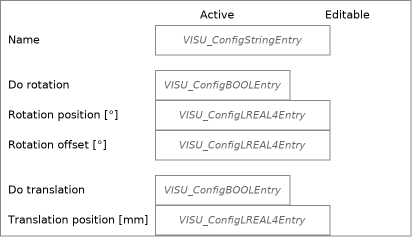
VISUALIZATION VISU_M3Config_KnownPosition  // 412x237
VAR_IN_OUT
	active : M3PositionConfig;
	editable : M3PositionConfig;
END_VAR
    Label (155,5 125x20), "Active"
    Label (285,5 125x20), "Editable"
    Label (5,25 125x30), "Name"
    Frame (155,25 175x30)
        shows VISU_ConfigStringEntry(active := active.name, editable := editable.name)
    Label (5,70 125x30), "Do rotation"
    Frame (155,70 135x30)
        shows VISU_ConfigBOOLEntry(active := active.doRotation, editable := editable.doRotation)
    Frame (155,100 175x30)
        shows VISU_ConfigLREAL4Entry(active := active.rotationPosition, editable := editable.rotationPosition)
    Label (5,100 125x30), "Rotation position [°]"
    Label (5,130 125x30), "Rotation offset [°]"
    Frame (155,130 175x30)
        shows VISU_ConfigLREAL4Entry(active := active.rotationOffset, editable := editable.rotationOffset)
    Label (5,175 125x30), "Do translation"
    Frame (155,175 135x30)
        shows VISU_ConfigBOOLEntry(active := active.doTranslation, editable := editable.doTranslation)
    Frame (155,205 175x30)
        shows VISU_ConfigLREAL4Entry(active := active.translationPosition, editable := editable.translationPosition)
    Label (5,205 150x30), "Translation position [mm]"
END_VISUALIZATION

(* stored: Version 1.1.0.1, ProductVersion 3.1.4019.2
   Visu VISU_M3Config_KnownPosition: Id {3b515ea5-8c9c-4e39-b443-8df539f7f9d6} *)
